(* PLC project my_app, Dassault Systèmes ControlBuild 2024x Refresh1 *)
(* stored: creationDateTime 2024-03-13T17:22:31-01:00 *)

PROGRAM sub
  VAR_INPUT
    entree : BOOL := false;
    entree2 : BOOL := false;
    entree3 : BOOL := false;
    entree4 : BOOL := false;
  END_VAR

(* FBD diagram, written out as Structured Text *)
END_PROGRAM

PROGRAM my_app.my_app
  VAR_INPUT
    entree : BOOL := false;
  END_VAR

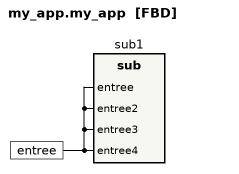
(* FBD diagram, written out as Structured Text *)
sub1(entree := entree, entree2 := entree, entree3 := entree, entree4 := entree);
END_PROGRAM
